// TIA Portal V15.1 export
// export: Created 2019-08-14T06:25:23.2499548Z, ExportSetting None, DisplayName Totally Integrated Automation Portal, DisplayVersion V15.1, DisplayName TIA Portal Openness, DisplayVersion V15.1, DisplayName STEP 7 Professional, DisplayVersion V15.1, DisplayName STEP 7 Safety, DisplayVersion V15.1, DisplayName WinCC Advanced, DisplayVersion V15.1
FUNCTION_BLOCK "#SKILL_NAME#_GetResult"   // FB15, SCL
{ S7_Optimized_Access := 'TRUE' }
// stored: MemoryReserve 100, SetENOAutomatically False
   VAR_INPUT
      Automatic : Bool;
   END_VAR
   VAR_OUTPUT
      Done : Bool;
   END_VAR
   VAR_IN_OUT
      ResultFeched : Bool;
      ResultTrigger : DInt;
      Parameter_Out : "type#SKILL_NAME#GetResultParameter_Out";
   END_VAR
   VAR
      OPC_UA_ServerMethodPre_Instance : OPC_UA_ServerMethodPre;
      OPC_UA_ServerMethodPost_Instance : OPC_UA_ServerMethodPost;
      UAMethod_OutParameters : "type#SKILL_NAME#GetResultParameter_Out";
      UAMethod : "UA_Method_Handle";
   END_VAR
BEGIN
   REGION PRE
       IF #UAMethod.Started = FALSE AND #UAMethod.Finished = FALSE THEN

           #OPC_UA_ServerMethodPre_Instance(Busy => #UAMethod.Pre.Busy,
                                            Done => #UAMethod.Pre.Done,
                                            Status => #UAMethod.Pre.Status,
                                            Error => #UAMethod.Pre.Error,
                                            UAMethod_Called => #UAMethod.Called);

           IF #UAMethod.Pre.Error THEN
               #UAMethod.ErrorMessage := WString#'Error at OPC_UA_ServerMethodPre';
           END_IF;

           IF #UAMethod.Pre.Done AND #UAMethod.Called THEN
               #UAMethod.Started := TRUE;
               #UAMethod.ErrorMessage := WString#'';
           END_IF;

       END_IF;

   END_REGION


   REGION FUNCTIONALITY 

       IF #UAMethod.Started = TRUE THEN
           #Done := FALSE;
           (*// 
           // User Code here
           //*)
           ;

           // submit result parameter from main skill FB
           // parameter is skill dependent
           #UAMethod_OutParameters := #Parameter_Out;

           #UAMethod.Result := 16#0;
           #UAMethod.ErrorMessage := WString#'';

           #UAMethod.Finished := TRUE;
           #UAMethod.Started := FALSE;
           #ResultFeched := TRUE;
       END_IF;

   END_REGION


   REGION POST
       IF #UAMethod.Finished = TRUE THEN
           #Done := TRUE;

           #OPC_UA_ServerMethodPost_Instance(UAMethod_Result := #UAMethod.Result,
                                             UAMethod_Finished := #UAMethod.Finished,
                                             Busy => #UAMethod.Post.Busy,
                                             Done => #UAMethod.Post.Done,
                                             Error => #UAMethod.Post.Error,
                                             Status => #UAMethod.Post.Status,
                                             UAMethod_OutParameters := #UAMethod_OutParameters);

           IF #UAMethod.Post.Error = TRUE THEN
               #UAMethod.ErrorMessage := WString#'Error at OPC_UA_ServerMethodPost';
               #UAMethod.Finished := FALSE;
           END_IF;

           IF #UAMethod.Post.Done = TRUE THEN
               #UAMethod.Finished := FALSE;
           END_IF;

       END_IF;

   END_REGION
END_FUNCTION_BLOCK
